// TIA Portal V18 export
// export: Created 2026-01-09T11:23:29.7823841Z, ExportSetting WithDefaults, DisplayName Totally Integrated Automation Portal, DisplayVersion V18 Update 5, DisplayName TIA Portal Openness, DisplayVersion V18 Update 5, DisplayName TIA Portal Teamcenter Gateway, DisplayVersion V18, DisplayName TIA Portal Version Control Interface, DisplayVersion V18, DisplayName SINAMICS Startdrive Advanced, DisplayVersion V18 SP2 Update 1, DisplayName SINAMICS Startdrive G110M, G120, G120C, G120D, G120P, G115D, DisplayVersion V18 SP2 Update 1, DisplayName SINAMICS Startdrive G130, G150, S120, S150, SINAMICS MV, S210, G220, S200, DisplayVersion V18 SP2 Update 1, DisplayName STEP 7 Professional, DisplayVersion V18 Update 5, DisplayName STEP 7 Safety, DisplayVersion V18, DisplayName WinCC Professional, DisplayVersion V18 Update 5
Screen "213 Scanner_801A1"  1280x800, Number=213, Template=02ManualUnit1
  ScreenLayer "Layer_0"
    FaceplateInstance "RCS_fpKeyenceSR1000_TP1200_1" at 30,148 size 1102x383  FaceplateTypeName=KeyenceSR1000@$@03_FacePlate@$@RCS_fpKeyenceSR1000_TP1200 V 0.0.8
      InterfacePropertyText "文本"  Text="801A1_ShafeScan / 801A1"
      Property := KeyenceSR1000Ctrl_801A1DB_sHMI
    Button "btnMenu5" at 512,725 size 128x75  Mode=Text, TextOff="A-读码器 801A1 / A-CodeReader 801A1", TextOn="A-读码器 801A1 / A-CodeReader 801A1"
      on Click: ActivateScreen(Screen name := , Object number := 0)
    Button "btnMenu4" at 384,725 size 128x75  Mode=Text, TextOff="A-伺服 381A1 / A-Servo 381A1", TextOn="A-伺服 381A1 / A-Servo 381A1"
      on Click: ActivateScreen(Screen name := 212-Servo_381A1, Object number := 0)
    Button "btnMenu6" at 640,725 size 128x75  Mode=Text, TextOff="A-读码器 804A1 / A-CodeReader 804A1", TextOn="A-读码器 804A1 / A-CodeReader 804A1"
      on Click: ActivateScreen(Screen name := 214 Scanner_804A1, Object number := 0)
    Button "btnMenu7" at 896,725 size 128x75  Mode=Text
    Button "btnMenu6_1" at 768,725 size 128x75  Mode=Text, TextOff="A-读码器 800A1 / A-CodeReader 800A1", TextOn="A-读码器 800A1 / A-CodeReader 800A1"
      on Click: ActivateScreen(Screen name := 215 X80Scanner_800A1, Object number := 0)
    Button "btnMenu7_1" at 1024,725 size 128x75  Mode=Text, TextOff="下一页 / NextPage", TextOn="下一页 / NextPage"
      on Click: ActivateScreen(Screen name := 216_Cylinder_A2, Object number := 0)
    Button "btnMenu4_1" at 256,725 size 128x75  Mode=Text, TextOff="A-伺服 380A1 / A-Servo 380A1", TextOn="A-伺服 380A1 / A-Servo 380A1"
      on Click: ActivateScreen(Screen name := 211-Servo_380A1, Object number := 0)
    Button "按钮_1" at 128,725 size 128x75  Mode=Text, PictureOff=向右箭头_0, TextOff="A-气缸1 / A-Cylinder1", TextOn="A-气缸1 / A-Cylinder1"
      on Click: ActivateScreen(Screen name := 210_Cylinder_A1, Object number := 0)
